{attribute addProperty BoxType "EL4712--0000"}
{attribute addProperty Id "Ch1_CycleCountAT %Q*Ch1_CycleCount_B92764D41620Ch1_SampleAT %Q*ARRAY[0..9] OF Ch1_Sample_4E940676160200Ch2_CycleCountAT %Q*Ch2_CycleCount_EB7284BC1620Ch2_SampleAT %Q*ARRAY[0..9] OF Ch2_Sample_50B89E9D160200WcStateAT %I*WcState_64F6A8C6810InfoDataAT %I*InfoData_7231B2DD80100"}
{attribute addProperty CRC "3612032114"}
{attribute addProperty SizeInBites "440"}
{attribute addProperty SizeInBytes "55"}
TYPE EL4712_C8B4D13D :
STRUCT
	{attribute addProperty Name "Ch1_CycleCount"}
	Ch1_CycleCount : Ch1_CycleCount_B92764D4;
	{attribute addProperty Name "Ch1_Sample"}
	Ch1_Sample : ARRAY[0..9] OF Ch1_Sample_4E940676;
	{attribute addProperty Name "Ch2_CycleCount"}
	Ch2_CycleCount : Ch2_CycleCount_EB7284BC;
	{attribute addProperty Name "Ch2_Sample"}
	Ch2_Sample : ARRAY[0..9] OF Ch2_Sample_50B89E9D;
	{attribute addProperty Name "WcState"}
	WcState : WcState_64F6A8C6;
	{attribute addProperty Name "InfoData"}
	InfoData : InfoData_7231B2DD;
END_STRUCT
END_TYPE

(* stored: Version 1.2.0.0, ProductVersion 3.1.4024.9
   DUT EL4712_C8B4D13D: Id {a4291c27-a141-4ef8-afe6-c3f691662ea2} *)
